// TIA Portal V20 export
// export: Created 2025-12-01T14:56:17.5716083Z, ExportSetting None, DisplayName Totally Integrated Automation Portal, DisplayVersion V20 Update 3, DisplayName TIA Portal Openness, DisplayVersion V20 Update 3, DisplayName TIA Portal Version Control Interface, DisplayVersion V20 Update 3, DisplayName STEP 7 Professional, DisplayVersion V20 Update 3, DisplayName STEP 7 Safety, DisplayVersion V20 Update 2, DisplayName WinCC Basic/Comfort/Advanced, DisplayVersion V20 Update 3, DisplayName WinCC Professional, DisplayVersion V20 Update 3, DisplayName WinCC Unified, DisplayVersion V20 Update 3
TYPE "InterlocK_UlmaQubiqa"
   STRUCT
      CCS_Online { ExternalVisible := 'False'} : Bool;
      CCS_Alive { ExternalVisible := 'False'} : Bool;
      CCS1_Run { ExternalVisible := 'False'} : Bool;
      CCS2_Run { ExternalVisible := 'False'} : Bool;
      CCS1_StartButton { ExternalVisible := 'False'} : Bool;
      CCS1_StopButton { ExternalVisible := 'False'} : Bool;
      CCS1_ResetButton { ExternalVisible := 'False'} : Bool;
      CCS2_StartButton { ExternalVisible := 'False'} : Bool;
      CCS2_StopButton { ExternalVisible := 'False'} : Bool;
      CCS2_ResetButton { ExternalVisible := 'False'} : Bool;
      ReserveOut_1_2 { ExternalVisible := 'False'} : Bool;
      ReserveOut_1_3 { ExternalVisible := 'False'} : Bool;
      ReserveOut_1_4 { ExternalVisible := 'False'} : Bool;
      ReserveOut_1_5 { ExternalVisible := 'False'} : Bool;
      ReserveOut_1_6 { ExternalVisible := 'False'} : Bool;
      ReserveOut_1_7 { ExternalVisible := 'False'} : Bool;
      RdyToReceive_L1 { ExternalVisible := 'False'} : Bool;   // Request to deliver a item to the tray loader from the manual line
      QueueCSSSorter_L1 { ExternalVisible := 'False'} : Bool;
      ReserveOut_2_2 { ExternalVisible := 'False'} : Bool;
      ReserveOut_2_3 { ExternalVisible := 'False'} : Bool;
      ReserveOut_2_4 { ExternalVisible := 'False'} : Bool;
      ReserveOut_2_5 { ExternalVisible := 'False'} : Bool;
      ReserveOut_2_6 { ExternalVisible := 'False'} : Bool;
      OrderFinished_Ok_L1 { ExternalVisible := 'False'} : Bool;
      StackRdy_Small_L1 { ExternalVisible := 'False'} : Bool;
      reservaOut_3_1 { ExternalVisible := 'False'} : Bool;
      reservaOut_3_2 { ExternalVisible := 'False'} : Bool;
      reservaOut_3_3 { ExternalVisible := 'False'} : Bool;
      reservaOut_3_4 { ExternalVisible := 'False'} : Bool;
      reservaOut_3_5 { ExternalVisible := 'False'} : Bool;
      reservaOut_3_6 { ExternalVisible := 'False'} : Bool;
      reservaOut_3_7 { ExternalVisible := 'False'} : Bool;
      Available_Small_L1 { ExternalVisible := 'False'} : Byte;
      StackRdy_Large_L1 { ExternalVisible := 'False'} : Bool;
      reservaOut_5_1 { ExternalVisible := 'False'} : Bool;
      reservaOut_5_2 { ExternalVisible := 'False'} : Bool;
      reservaOut_5_3 { ExternalVisible := 'False'} : Bool;
      reservaOut_5_4 { ExternalVisible := 'False'} : Bool;
      reservaOut_5_5 { ExternalVisible := 'False'} : Bool;
      reservaOut_5_6 { ExternalVisible := 'False'} : Bool;
      reservaOut_5_7 { ExternalVisible := 'False'} : Bool;
      Available_Large_L1 { ExternalVisible := 'False'} : Byte;
      RequestTodeliver_L1 { ExternalVisible := 'False'} : Bool;
      reservaOut_7_1 { ExternalVisible := 'False'} : Bool;
      OrderFinished_L1 { ExternalVisible := 'False'} : Bool;
      reservaOut_7_3 { ExternalVisible := 'False'} : Bool;
      reservaOut_7_4 { ExternalVisible := 'False'} : Bool;
      reservaOut_7_5 { ExternalVisible := 'False'} : Bool;
      reservaOut_7_6 { ExternalVisible := 'False'} : Bool;
      reservaOut_7_7 { ExternalVisible := 'False'} : Bool;
      ItemsNo_L1 { ExternalVisible := 'False'} : Int;
      ItemsNoTotal_L1 { ExternalVisible := 'False'} : Int;
      Length_PID_L1 { ExternalVisible := 'False'} : Int;
      PID_L1 { ExternalVisible := 'False'} : Array[0..19] of Char;
      RdyToReceive_L2 { ExternalVisible := 'False'} : Bool;
      QueueCCSSorter_L2 { ExternalVisible := 'False'} : Bool;
      ReserveOut_50_2 { ExternalVisible := 'False'} : Bool;
      ReserveOut_50_3 { ExternalVisible := 'False'} : Bool;
      ReserveOut_50_4 { ExternalVisible := 'False'} : Bool;
      ReserveOut_50_5 { ExternalVisible := 'False'} : Bool;
      ReserveOut_50_6 { ExternalVisible := 'False'} : Bool;
      OrderFinished_Ok_L2 { ExternalVisible := 'False'} : Bool;
      StackRdy_Small_L2 { ExternalVisible := 'False'} : Bool;
      reservaOut_51_1 { ExternalVisible := 'False'} : Bool;
      reservaOut_51_2 { ExternalVisible := 'False'} : Bool;
      reservaOut_51_3 { ExternalVisible := 'False'} : Bool;
      reservaOut_51_4 { ExternalVisible := 'False'} : Bool;
      reservaOut_51_5 { ExternalVisible := 'False'} : Bool;
      reservaOut_51_6 { ExternalVisible := 'False'} : Bool;
      reservaOut_51_7 { ExternalVisible := 'False'} : Bool;
      Available_Small_L2 { ExternalVisible := 'False'} : Byte;
      StackRdy_Large_L2 { ExternalVisible := 'False'} : Bool;
      reservaOut_53_1 { ExternalVisible := 'False'} : Bool;
      reservaOut_53_2 { ExternalVisible := 'False'} : Bool;
      reservaOut_53_3 { ExternalVisible := 'False'} : Bool;
      reservaOut_53_4 { ExternalVisible := 'False'} : Bool;
      reservaOut_53_5 { ExternalVisible := 'False'} : Bool;
      reservaOut_53_6 { ExternalVisible := 'False'} : Bool;
      reservaOut_53_7 { ExternalVisible := 'False'} : Bool;
      Available_Large_L2 { ExternalVisible := 'False'} : Byte;
      RequestToDeliver_L2 { ExternalVisible := 'False'} : Bool;
      ReserveOut_55_2 { ExternalVisible := 'False'} : Bool;
      OrderFinished_L2 { ExternalVisible := 'False'} : Bool;
      ReserveOut_55_3 { ExternalVisible := 'False'} : Bool;
      ReserveOut_55_4 { ExternalVisible := 'False'} : Bool;
      ReserveOut_55_5 { ExternalVisible := 'False'} : Bool;
      ReserveOut_55_6 { ExternalVisible := 'False'} : Bool;
      ReserveOut_55_7 { ExternalVisible := 'False'} : Bool;
      ItemsNo_L2 { ExternalVisible := 'False'} : Int;
      ItemsNoTotal_L2 { ExternalVisible := 'False'} : Int;
      Length_PID_L2 { ExternalVisible := 'False'} : Int;
      PID_L2 { ExternalVisible := 'False'} : Array[0..19] of Char;
   END_STRUCT;
END_TYPE
